// TIA Portal V20 export
FUNCTION_BLOCK "MotionTemp"   // FB142, SCL
{ S7_Optimized_Access := 'TRUE' }
// stored: MemoryReserve 100, SetENOAutomatically false
   VAR
      mcPower { S7_SetPoint := 'True'} : Array[1..50] of MC_POWER;
      mcHome { S7_SetPoint := 'True'} : Array[1..50] of MC_HOME;
      statOn { S7_SetPoint := 'True'} : Bool;
      instServoOnTriggerr : R_TRIG;
   END_VAR
   VAR_TEMP
      i : DInt;
   END_VAR
BEGIN

   #instServoOnTriggerr(CLK:=#statOn);

   IF #instServoOnTriggerr.Q THEN
       #mcPower[1].Enable := TRUE;
       #mcPower[2].Enable := TRUE;
       #mcPower[3].Enable := TRUE;
       #mcPower[4].Enable := TRUE;
       #mcPower[5].Enable := TRUE;
       #mcPower[6].Enable := TRUE;
       #mcPower[7].Enable := TRUE;
       #mcPower[8].Enable := TRUE;
       #mcPower[9].Enable := TRUE;
       #mcPower[10].Enable := TRUE;
       #mcPower[11].Enable := TRUE;
       #mcPower[12].Enable := TRUE;
       #mcPower[13].Enable := TRUE;
       #mcPower[14].Enable := TRUE;
       #mcHome[1].Execute := TRUE;
       #mcHome[2].Execute := TRUE;
       #mcHome[3].Execute := TRUE;
       #mcHome[4].Execute := TRUE;
       #mcHome[5].Execute := TRUE;
       #mcHome[6].Execute := TRUE;
       #mcHome[7].Execute := TRUE;
       #mcHome[8].Execute := TRUE;
       #mcHome[9].Execute := TRUE;
       #mcHome[10].Execute := TRUE;
       #mcHome[11].Execute := TRUE;
       #mcHome[12].Execute := TRUE;
       #mcHome[13].Execute := TRUE;
       #mcHome[14].Execute := TRUE;

   END_IF;

   #mcPower[1](Axis:="BA010AZCR_MasterVirtualAxis");
   #mcHome[1](Axis := "BA010AZCR_MasterVirtualAxis");

   #mcPower[2](Axis := "BA010AZCR_UnwinderVirtualAxis");
   #mcHome[2](Axis := "BA010AZCR_UnwinderVirtualAxis");

   #mcPower[3](Axis := "BA010AZCR_ConveyorVirtualAxis");
   #mcHome[3](Axis := "BA010AZCR_ConveyorVirtualAxis");

   #mcPower[4](Axis := "BA010AZCRDR1_UnwinderLeftAxisB");
   #mcHome[4](Axis := "BA010AZCRDR1_UnwinderLeftAxisB");

   #mcPower[5](Axis := "BA010AZCRDR3_CompensatorAxisZ");
   #mcHome[5](Axis := "BA010AZCRDR3_CompensatorAxisZ");

   #mcPower[6](Axis := "BA010AZCRDR4_FeedingRollAxisB");
   #mcHome[6](Axis := "BA010AZCRDR4_FeedingRollAxisB");

   #mcPower[7](Axis := "BA010AZCRDR5_ElectordCutterAxisZ");
   #mcHome[7](Axis := "BA010AZCRDR5_ElectordCutterAxisZ");

   #mcPower[8](Axis := "BA010AZCRDR9_VisionAxisZ");
   #mcHome[8](Axis := "BA010AZCRDR9_VisionAxisZ");

   #mcPower[9](Axis := "BA010AZCRDR10_NgKickerAxisZ");
   #mcHome[9](Axis := "BA010AZCRDR10_NgKickerAxisZ");

   #mcPower[10](Axis := "BA010AZCRDR11_PassKickerAxisZ");
   #mcHome[10](Axis := "BA010AZCRDR11_PassKickerAxisZ");

   #mcPower[11](Axis := "BA010AZCRDR12_CutConveyorAxisB");
   #mcHome[11](Axis := "BA010AZCRDR12_CutConveyorAxisB");

   #mcPower[12](Axis := "BA010AZCRDR13_NgConveyorAxisB");
   #mcHome[12](Axis := "BA010AZCRDR13_NgConveyorAxisB");

   #mcPower[13](Axis := "BA010AZCRDR14_Stack1ConveyorAxisB");
   #mcHome[13](Axis := "BA010AZCRDR14_Stack1ConveyorAxisB");

   #mcPower[14](Axis := "BA010AZCRDR15_Stack2ConveyorAxisB");
   #mcHome[14](Axis := "BA010AZCRDR15_Stack2ConveyorAxisB");
END_FUNCTION_BLOCK
